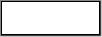
VISUALIZATION VISU_SubSubSystemButton  // 102x37
VAR_IN_OUT
    widget : SubSubSystemButtonWidget;
END_VAR
    Rectangle (0,0 100x35), invisible if: widget.isNotOrange
    Rectangle (0,0 100x35), invisible if: widget.isNotGray
    Rectangle (0,0 100x35), invisible if: widget.isNotBlue
    Rectangle (0,0 100x35), invisible if: widget.isNotRed
    Rectangle (0,0 100x35), invisible if: widget.isNotGreen
    Rectangle (0,0 100x35), "%s", text variable: widget.name
    Rectangle (0,0 100x35), invisible if: widget.notActivated
    Line (0,34) (100,34), invisible if: widget.activated
    Line (99,0) (99,35), invisible if: widget.activated
    Line (98,0) (0,0), invisible if: widget.activated
    Line (0,35) (0,0), invisible if: widget.activated
    Line (100,35) (100,1), invisible if: widget.notActivated
    Line (0,1) (99,1), invisible if: widget.notActivated
    Line (1,0) (1,35), invisible if: widget.notActivated
    Line (100,35) (1,35), invisible if: widget.notActivated
END_VISUALIZATION

(* stored: Version 1.1.0.1, ProductVersion 3.1.4019.2
   Visu VISU_SubSubSystemButton: Id {2c5d5b18-563f-4c54-8191-363734449b62} *)
